TYPE ST_CoeEntry_UINT EXTENDS ST_CoeEntry :
STRUCT
	Value	: UINT;
END_STRUCT
END_TYPE

(* stored: Version 1.1.0.1, ProductVersion 3.1.4024.13
   DUT ST_CoeEntry_UINT: Id {577770cf-1335-0de1-1e88-95460d04421a} *)
